// TIA Portal V18 export
// export: Created 2000-01-01T00:00:00.0000000Z, ExportSetting None
FUNCTION_BLOCK "FB_Motor"   // FB, LAD
BEGIN

REGION Network 1: Start latch
   // Start stop latch parser fixture
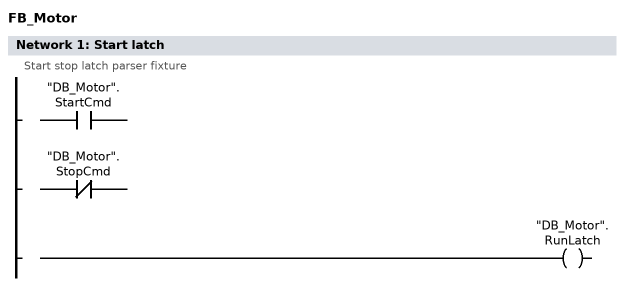
   "DB_Motor".RunLatch := TRUE;
END_REGION
END_FUNCTION_BLOCK
